// Incremental Sparkplug B payload builder.
//
// Wraps FB_ProtoWriter with Sparkplug-aware metric write methods. The caller
// provides an external buffer so payload capacity can be sized appropriately
// for the message type (large for NBIRTH/DBIRTH, small for DDATA).
//
// Usage:
//   fbPayload.Init(pBuffer, nCapacity);
//   fbPayload.WriteHeader(nTimestamp, nSeq);
//   fbPayload.WriteBoolMetric('MotorRunning', 1, E_SparkplugDataType.Boolean, TRUE);
//   fbPayload.WriteUInt32Metric('', 2, E_SparkplugDataType.UInt32, nSpeed);  // DATA mode: no name
//   // publish fbPayload.Buffer for fbPayload.Length bytes
//
// Metric name conventions:
//   BIRTH messages  — pass the metric name; alias is also included for future DATA messages.
//   DATA messages   — pass sName := '' to omit the name and use alias only (saves bandwidth).
//   System metrics  — pass nAlias := 0 to omit the alias field (name-only, e.g. bdSeq).
FUNCTION_BLOCK FB_SparkplugPayload
VAR
	_fbPayload		: FB_ProtoWriter;				// outer Payload message
	_fbMetric		: FB_ProtoWriter;				// inner Metric message (reused per metric)
	_aBufMetric		: ARRAY[0..511] OF BYTE;		// temp buffer for one encoded Metric
END_VAR

// FB body intentionally empty — all logic is in the methods below.

// Binds the payload builder to an external buffer and resets it.
// Must be called before any Write methods.
METHOD Init
VAR_INPUT
	pBuffer		: POINTER TO BYTE;
	nCapacity	: UDINT;
END_VAR
_fbPayload.Init(pBuffer, nCapacity);
END_METHOD

// Resets the write position without re-binding the buffer.
// Use when re-encoding into the same buffer (e.g. periodic DDATA).
METHOD Reset
_fbPayload.Reset();
END_METHOD

// Writes the Payload-level timestamp (field 1) and seq (field 4).
// Must be the first Write call after Init/Reset.
//
// Sparkplug field numbers for Payload (from sparkplug_b.proto):
//   1 = timestamp (uint64, ms since Unix epoch)
//   2 = metrics   (repeated, length-delimited)
//   3 = seq       (uint64, 0–255 wrapping)
//   4 = uuid      (string — not used by this library)
METHOD WriteHeader : BOOL
VAR_INPUT
	nTimestamp	: ULINT;
	nSeq		: ULINT;
END_VAR
WriteHeader := _fbPayload.WriteUInt64(1, nTimestamp)
	AND _fbPayload.WriteUInt64(3, nSeq);
END_METHOD

METHOD WriteBoolMetric : BOOL
VAR_INPUT
	sName		: STRING(255);
	nAlias		: ULINT;
	eDataType	: E_SparkplugDataType;
	bValue		: BOOL;
END_VAR
_fbMetric.Init(ADR(_aBufMetric), SIZEOF(_aBufMetric));
IF LEN(sName) > 0  THEN _fbMetric.WriteString(1, sName); END_IF
IF nAlias > 0      THEN _fbMetric.WriteUInt64(2, nAlias); END_IF
_fbMetric.WriteUInt32(4, TO_UDINT(eDataType));
_fbMetric.WriteBool(14, bValue);
WriteBoolMetric := _fbPayload.WriteBytes(2, ADR(_aBufMetric), _fbMetric.Length);
END_METHOD

// For Int8, Int16, Int32, UInt8, UInt16, UInt32 — encoded in proto field 10 (int_value).
METHOD WriteUInt32Metric : BOOL
VAR_INPUT
	sName		: STRING(255);
	nAlias		: ULINT;
	eDataType	: E_SparkplugDataType;
	nValue		: UDINT;
END_VAR
_fbMetric.Init(ADR(_aBufMetric), SIZEOF(_aBufMetric));
IF LEN(sName) > 0  THEN _fbMetric.WriteString(1, sName); END_IF
IF nAlias > 0      THEN _fbMetric.WriteUInt64(2, nAlias); END_IF
_fbMetric.WriteUInt32(4, TO_UDINT(eDataType));
_fbMetric.WriteUInt32(10, nValue);
WriteUInt32Metric := _fbPayload.WriteBytes(2, ADR(_aBufMetric), _fbMetric.Length);
END_METHOD

// For Int64, UInt64, DateTime — encoded in proto field 11 (long_value).
METHOD WriteUInt64Metric : BOOL
VAR_INPUT
	sName		: STRING(255);
	nAlias		: ULINT;
	eDataType	: E_SparkplugDataType;
	nValue		: ULINT;
END_VAR
_fbMetric.Init(ADR(_aBufMetric), SIZEOF(_aBufMetric));
IF LEN(sName) > 0  THEN _fbMetric.WriteString(1, sName); END_IF
IF nAlias > 0      THEN _fbMetric.WriteUInt64(2, nAlias); END_IF
_fbMetric.WriteUInt32(4, TO_UDINT(eDataType));
_fbMetric.WriteUInt64(11, nValue);
WriteUInt64Metric := _fbPayload.WriteBytes(2, ADR(_aBufMetric), _fbMetric.Length);
END_METHOD

METHOD WriteFloatMetric : BOOL
VAR_INPUT
	sName		: STRING(255);
	nAlias		: ULINT;
	eDataType	: E_SparkplugDataType;
	fValue		: REAL;
END_VAR
_fbMetric.Init(ADR(_aBufMetric), SIZEOF(_aBufMetric));
IF LEN(sName) > 0  THEN _fbMetric.WriteString(1, sName); END_IF
IF nAlias > 0      THEN _fbMetric.WriteUInt64(2, nAlias); END_IF
_fbMetric.WriteUInt32(4, TO_UDINT(eDataType));
_fbMetric.WriteFloat(12, fValue);
WriteFloatMetric := _fbPayload.WriteBytes(2, ADR(_aBufMetric), _fbMetric.Length);
END_METHOD

METHOD WriteDoubleMetric : BOOL
VAR_INPUT
	sName		: STRING(255);
	nAlias		: ULINT;
	eDataType	: E_SparkplugDataType;
	fValue		: LREAL;
END_VAR
_fbMetric.Init(ADR(_aBufMetric), SIZEOF(_aBufMetric));
IF LEN(sName) > 0  THEN _fbMetric.WriteString(1, sName); END_IF
IF nAlias > 0      THEN _fbMetric.WriteUInt64(2, nAlias); END_IF
_fbMetric.WriteUInt32(4, TO_UDINT(eDataType));
_fbMetric.WriteDouble(13, fValue);
WriteDoubleMetric := _fbPayload.WriteBytes(2, ADR(_aBufMetric), _fbMetric.Length);
END_METHOD

// For String, Text, UUID data types.
METHOD WriteStringMetric : BOOL
VAR_INPUT
	sName		: STRING(255);
	nAlias		: ULINT;
	eDataType	: E_SparkplugDataType;
	sValue		: STRING(255);
END_VAR
_fbMetric.Init(ADR(_aBufMetric), SIZEOF(_aBufMetric));
IF LEN(sName) > 0  THEN _fbMetric.WriteString(1, sName); END_IF
IF nAlias > 0      THEN _fbMetric.WriteUInt64(2, nAlias); END_IF
_fbMetric.WriteUInt32(4, TO_UDINT(eDataType));
_fbMetric.WriteString(15, sValue);
WriteStringMetric := _fbPayload.WriteBytes(2, ADR(_aBufMetric), _fbMetric.Length);
END_METHOD

// Pointer to the start of the encoded payload. Valid until the next Init call.
PROPERTY Buffer : POINTER TO BYTE
GET
Buffer := _fbPayload.Buffer;
END_GET
END_PROPERTY

PROPERTY Length : UDINT
GET
Length := _fbPayload.Length;
END_GET
END_PROPERTY

PROPERTY HasError : BOOL
GET
HasError := _fbPayload.HasError;
END_GET
END_PROPERTY

END_FUNCTION_BLOCK

(* stored: Version 1.1.0.1
   POU FB_SparkplugPayload: Id {11111111-2222-3333-4444-555555555555}, SpecialFunc None
   Method Init: Id {aaaaaaaa-bbbb-cccc-dddd-000000000001}
   Method Reset: Id {aaaaaaaa-bbbb-cccc-dddd-000000000002}
   Method WriteHeader: Id {aaaaaaaa-bbbb-cccc-dddd-000000000003}
   Method WriteBoolMetric: Id {aaaaaaaa-bbbb-cccc-dddd-000000000010}
   Method WriteUInt32Metric: Id {aaaaaaaa-bbbb-cccc-dddd-000000000011}
   Method WriteUInt64Metric: Id {aaaaaaaa-bbbb-cccc-dddd-000000000012}
   Method WriteFloatMetric: Id {aaaaaaaa-bbbb-cccc-dddd-000000000013}
   Method WriteDoubleMetric: Id {aaaaaaaa-bbbb-cccc-dddd-000000000014}
   Method WriteStringMetric: Id {aaaaaaaa-bbbb-cccc-dddd-000000000015}
   Property Buffer: Id {aaaaaaaa-bbbb-cccc-dddd-000000000020}
   Get Get: Id {aaaaaaaa-bbbb-cccc-dddd-000000000021}
   Property Length: Id {aaaaaaaa-bbbb-cccc-dddd-000000000022}
   Get Get: Id {aaaaaaaa-bbbb-cccc-dddd-000000000023}
   Property HasError: Id {aaaaaaaa-bbbb-cccc-dddd-000000000024}
   Get Get: Id {aaaaaaaa-bbbb-cccc-dddd-000000000025} *)
